FUNCTION_BLOCK fb_engageUndockAll
VAR_INPUT
END_VAR
VAR_OUTPUT
END_VAR
VAR
	step: INT;
	cleanin: fb_cleanIn;
	cleanout: fb_cleanOut;
	undock: fb_undock;
	dock: fb_dock;
	opcl: fb_dsopenclose;
END_VAR

CASE step OF
	0:
		IF Allengage.cleanOutu THEN
			cntrlstate.cleanout := FALSE;
			cleanout(done := cntrlstate.cleanout);
			IF cntrlstate.cleanout THEN
				Allengage.cleanOutu := FALSE;
				Allengage.stepper := TRUE;
				step := 1;
			END_IF
		END_IF
	1: 
		IF Allengage.stepper THEN
			DSin.open := TRUE;
			opcl();
			IF NOT DSin.open THEN
				step := 2;
				Allengage.undock := TRUE;
				Allengage.stepper := FALSE;
			END_IF
		END_IF
	
	2:
		IF Allengage.undock THEN
			cntrlstate.undock := FALSE;
			undock();
			IF cntrlstate.undock THEN
				Allengage.undock := FALSE;
				Allengage.stepper := TRUE;
				step := 3;
			END_IF
		END_IF
	
	3:
		IF Allengage.stepper THEN
			DSin.close := TRUE;
			opcl();
			IF NOT DSin.close THEN
				step := 4;
				Allengage.stepper := FALSE;
			END_IF
		END_IF
		
	4:
		engage.allundock := FALSE;
		step := 0;
END_CASE

END_FUNCTION_BLOCK

(* stored: Version 1.1.0.1, ProductVersion 3.1.4024.5
   POU fb_engageUndockAll: Id {64f8b081-bc4b-4875-b35b-36179f8cc1e5}, SpecialFunc None *)
